TYPE ELM3002InputwTimestamp :
STRUCT
	analogInput	:	LREAL;
	timestamp	:	ULINT;
END_STRUCT
END_TYPE

(* stored: Version 1.1.0.1, ProductVersion 3.1.4024.12
   DUT ELM3002InputwTimestamp: Id {9d378d13-e644-49ea-a1e3-2d0b716d3554} *)
